Universal Robots URScript: T005_qwen2.5-coder_32b_baseline_rep1.urscript

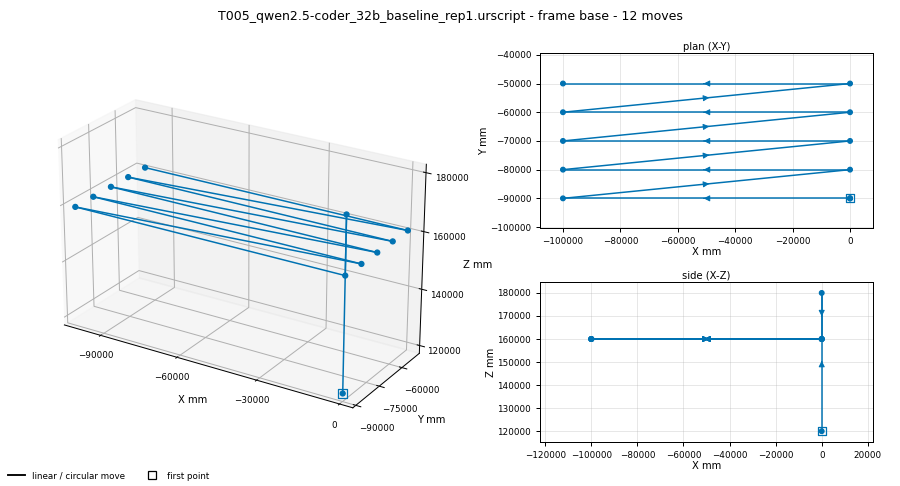
[picture p0: tool path of T005_qwen2.5-coder_32b_baseline_rep1.urscript in frame base, 12 of 12 moves have a stored position in this frame; points joined in program order, loops and branches not executed]
def visual_inspection_scan():
    # Move to home position
    movej(p[0, -90, 120, 0, -90, 0], a=1.4, v=1.05)

    # Approach inspection start position (above surface)
    movel(p[0, -90, 180, 0, -90, 0], a=1.2, v=1.02)

    # Descend to scan height (150 mm above part)
    movel(p[0, -90, 160, 0, -90, 0], a=1.2, v=0.8)

    # Scan line 1 — Y sweep
    movel(p[-100, -90, 160, 0, -90, 0], a=1.2, v=0.5)

    # Step to scan line 2 (+X)
    movel(p[0, -80, 160, 0, -90, 0], a=1.2, v=0.8)

    # Scan line 2 — Y sweep
    movel(p[-100, -80, 160, 0, -90, 0], a=1.2, v=0.5)

    # Step to scan line 3 (+X)
    movel(p[0, -70, 160, 0, -90, 0], a=1.2, v=0.8)

    # Scan line 3 — Y sweep
    movel(p[-100, -70, 160, 0, -90, 0], a=1.2, v=0.5)

    # Step to scan line 4 (+X)
    movel(p[0, -60, 160, 0, -90, 0], a=1.2, v=0.8)

    # Scan line 4 — Y sweep
    movel(p[-100, -60, 160, 0, -90, 0], a=1.2, v=0.5)

    # Step to scan line 5 (+X)
    movel(p[0, -50, 160, 0, -90, 0], a=1.2, v=0.8)

    # Scan line 5 — Y sweep
    movel(p[-100, -50, 160, 0, -90, 0], a=1.2, v=0.5)

end

visual_inspection_scan()
